// TIA Portal V17 export
// export: Created 2024-06-16T17:47:34.2368864Z, ExportSetting WithDefaults, DisplayName Totally Integrated Automation Portal, DisplayVersion V17, DisplayName TIA Portal Openness, DisplayVersion V17, DisplayName TIA Portal Version Control Interface, DisplayVersion V17, DisplayName STEP 7 Professional, DisplayVersion V17, DisplayName STEP 7 Safety, DisplayVersion V17, DisplayName WinCC Professional, DisplayVersion V17
DATA_BLOCK "St4_In"   // DB405
{ S7_Optimized_Access := 'TRUE' }
VERSION : 0.1
// stored: AutoNumber false, DBAccessibleFromOPCUA true, DBAccessibleFromWebserver true, IsOnlyStoredInLoadMemory false, IsRetainMemResEnabled false, IsWriteProtectedInAS false, MemoryReserve 100
   VAR
      Loquet_Haut : Bool;   // Loquet haut : Pas de déplacement barquette
      Cpt_M : Bool;   // Présence pile en zone de marquage
      PincesDC_Ouvert : Bool;   // Pinces de préhension Déchagement C : Ouverte
      PincesDC_Fermee : Bool;   // Pinces de préhension Déchagement C : Fermée
      Cpt_DC1 : Bool;   // Présence pile en zone Déchagement C1
      Cpt_DC2 : Bool;   // Présence pile en zone Déchagement : C2
      PoussoirC_Haut : Bool;   // Poussoir C en position : Haut
      PincesDNC_Ouvert : Bool;   // Pinces de préhension Déchagement NC : Ouverte
      PincesDNC_Fermee : Bool;   // Pinces de préhension Déchagement NC : Ferméee
      Cpt_DNC0 : Bool;   // Présence pile en zone Déchagement NC0
      Cpt_DNC1 : Bool;   // Présence pile en zone Déchagement DNC1
      Cpt_DNC2 : Bool;   // Présence pile en zone Déchagement DNC2
      PoussoirNC_Haut : Bool;   // Poussoir NC en position : Haut
   END_VAR
BEGIN
END_DATA_BLOCK
